Universal Robots PolyScope program: interpret.urp

Program interpret (installation=default directory=/programs/RemoteOperation createdIn=5.10.0.106268 lastSavedIn=5.10.0.106268 robotSerialNumber=20185500191)
Calibrated DH parameters: a=[0.000131, -0.165639, -0.102041, 0.000082, 0.000046, 0]; d=[0.162455, 220.258006, 1988.136334, -2208.260978, 0.099826, 0.099896]; alpha=[1.570482, -0.001777, -0.000172, 1.570393, -1.570735, 0]; deltaTheta=[0, -1.170526, -0.137148, 1.307669, -0.000001, 0]
Robot Program (runOnlyOnce=true)
  Script: interpreter_mode(clearQueueOnEnter=False)
